DEVICE_TYPE _TCREST
  (* Standard: 61499-2 *)
  (* Version 0.1, 2017-00-09, hpea485, UOA *)
  VAR_INPUT
    tcrestInput : BOOL;
    Core0Input : INT;
  END_VAR
  RESOURCE Resource : _Core0(Core0Input := 0)
  END_RESOURCE
  RESOURCE Resource1 : _Core1(Core1Input := 1)
  END_RESOURCE
END_DEVICE_TYPE
